Omron CX-Programmer project NewProject (CX-Programmer 9.42)

# PLC Industrial_Sorter: CJ1M CPU11
I/O table (CPU CJ1M-CPU11): rack 0 slot 0 CJ1W-ID211; rack 0 slot 1 CJ1W-ID211; rack 0 slot 2 CJ1W-OC211; rack 0 slot 3 CJ1W-MAD42

## Global symbols (name address type ; comment)
0.00 BOOL  ; Start
0.01 BOOL  ; Stop
W0.00 BOOL  ; Permissive

## Program NewProgram1 (cyclic task 0)

### Section Section1

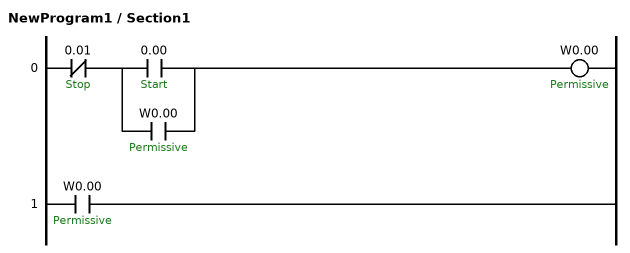
; rung 0
LDNOT 0.01  ; Stop
LD 0.00  ; Start
OR W0.00  ; Permissive
ANDLD
OUT W0.00  ; Permissive
; rung 1
LD W0.00  ; Permissive

### Section END
; rung 0
END(001)